// TIA Portal V16 export
// export: Created 2025-08-01T13:38:04.2195309Z, ExportSetting WithDefaults, DisplayName Totally Integrated Automation Portal, DisplayVersion V16, DisplayName TIA Portal Version Control Interface, DisplayVersion V16, DisplayName TIA Portal Openness, DisplayVersion V16, DisplayName STEP 7 Professional, DisplayVersion V16, DisplayName STEP 7 Safety, DisplayVersion V16, DisplayName WinCC Advanced, DisplayVersion V16
DATA_BLOCK "ProductBuffer_V2_DB"   // DB66
VERSION : 0.1
// stored: AutoNumber true, InstanceOfName ProductBuffer_V2, InstanceOfType FB
"ProductBuffer_V2"
   // VAR_INPUT
   //    SensorInput : Bool;
   //    SensorManual : Bool;
   //    TimeDelay : Time;
   //    SystemTime : Time;
   //    TriggerFeedback : Bool;
   // END_VAR
   // VAR_OUTPUT
   //    TriggerMovement : Bool;
   //    InsertIndex { ExternalVisible := 'False'; ExternalWritable := 'False'} : Int;
   //    ProductCount : Int;
   //    SystemTicks : DInt;
   // END_VAR
   // VAR RETAIN
   //    ProductQueue : Array[0..1] of "ProductEntry";
   //    StartTimes : Struct
   //       _0 : Time;
   //       _1 : Time;
   //       _2 : Time;
   //       _3 : Time;
   //       _4 : Time;
   //       _5 : Time;
   //       _6 : Time;
   //       _7 : Time;
   //       _8 : Time;
   //       _9 : Time;
   //    END_STRUCT;
   //    Actives : Struct
   //       _0 : Bool;
   //       _1 : Bool;
   //       _2 : Bool;
   //       _3 : Bool;
   //       _4 : Bool;
   //       _5 : Bool;
   //       _6 : Bool;
   //       _7 : Bool;
   //       _8 : Bool;
   //       _9 : Bool;
   //    END_STRUCT;
   //    PrevSensor { ExternalVisible := 'False'; ExternalWritable := 'False'} : Bool;
   //    MovementActive { ExternalVisible := 'False'; ExternalWritable := 'False'} : Bool;
   //    i { ExternalVisible := 'False'; ExternalWritable := 'False'} : Int;
   //    Elapsed { ExternalVisible := 'False'; ExternalWritable := 'False'} : DInt;
   // END_VAR
BEGIN
END_DATA_BLOCK
